PROGRAM POU_Persistent
VAR
	fbWritePersistentData: FB_WritePersistentData;
	bPersistentWr: BOOL;
	
END_VAR


fbWritePersistentData(
	NETID:= , 
	PORT:= 851 , 
	START:= bPersistentWr, 
	TMOUT:= , 
	MODE:= , 
	BUSY=> , 
	ERR=> , 
	ERRID=> );
	
bPersistentWr:= FALSE;

END_PROGRAM

(* stored: Version 1.1.0.1, ProductVersion 3.1.4024.12
   POU POU_Persistent: Id {e48eeb10-ca8b-4438-90d6-90fda42a3969}, SpecialFunc None *)
